// TIA Portal V20 export
DATA_BLOCK "IDB_Merging"   // DB30011
// stored: InstanceOfName EmptyLine.FB_Merging, InstanceOfType FB, Namespace EmptyLine
"EmptyLine.FB_Merging"
   // VAR
   //    "Merge_J1.2.4" { S7_SetPoint := 'True'} : "Global.FB_Merging";
   // END_VAR
BEGIN
END_DATA_BLOCK
